INTERFACE I_TempSens

METHOD Run : BOOL
VAR_INPUT
END_VAR
END_METHOD

PROPERTY Temperature : Real
GET
END_GET
SET
END_SET
END_PROPERTY

END_INTERFACE

(* stored: Version 1.1.0.1, ProductVersion 3.1.4022.10
   Itf I_TempSens: Id {0b304bd9-4067-4553-83b2-c039f01142f8}
   Method Run: Id {f05b2d95-0764-4ad5-9700-941d32d8d4da}
   Property Temperature: Id {ed04a6e5-b17b-4ab4-9023-ba82f62cd569}
   Get Get: Id {b1bc7acf-88e1-4c7e-b062-1787da4338fc}
   Set Set: Id {26a8fc85-3415-44fc-81c3-45dc46a2aff3} *)
